PROGRAM P1_04_Alarms
VAR
	iActive				:INT;
	iAck				:INT;
	iRaise				:INT;
	iDisabled			:INT;
	
	bAlarmDisabled		:BOOL;
	
	bAlarmActive		:BOOL;
	bSP_AlarmActive		:BOOL;
	TON_AlarmOK			:TON;
	TON_SP_AlarmOK		:TON;
END_VAR

VAR PERSISTENT
	fbAlarm				:ARRAY [0..69] OF FB_AlarmDiagnostic;
END_VAR

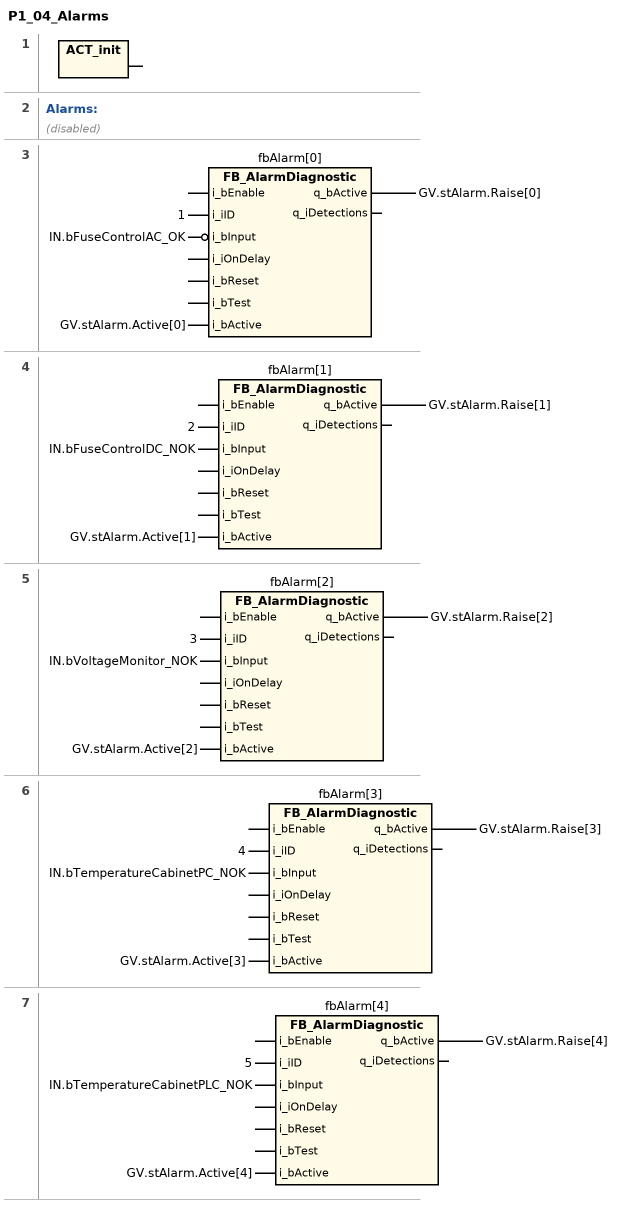
// NETWORK 1
ACT_init();

// NETWORK 2 (disabled)
// label: Alarms

// NETWORK 3
fbAlarm[0](i_iID := 1, i_bInput := NOT IN.bFuseControlAC_OK, i_bActive := GV.stAlarm.Active[0]); // FB_AlarmDiagnostic
GV.stAlarm.Raise[0] := fbAlarm[0].q_bActive;

// NETWORK 4
fbAlarm[1](i_iID := 2, i_bInput := IN.bFuseControlDC_NOK, i_bActive := GV.stAlarm.Active[1]); // FB_AlarmDiagnostic
GV.stAlarm.Raise[1] := fbAlarm[1].q_bActive;

// NETWORK 5
fbAlarm[2](i_iID := 3, i_bInput := IN.bVoltageMonitor_NOK, i_bActive := GV.stAlarm.Active[2]); // FB_AlarmDiagnostic
GV.stAlarm.Raise[2] := fbAlarm[2].q_bActive;

// NETWORK 6
fbAlarm[3](i_iID := 4, i_bInput := IN.bTemperatureCabinetPC_NOK, i_bActive := GV.stAlarm.Active[3]); // FB_AlarmDiagnostic
GV.stAlarm.Raise[3] := fbAlarm[3].q_bActive;

// NETWORK 7
fbAlarm[4](i_iID := 5, i_bInput := IN.bTemperatureCabinetPLC_NOK, i_bActive := GV.stAlarm.Active[4]); // FB_AlarmDiagnostic
GV.stAlarm.Raise[4] := fbAlarm[4].q_bActive;

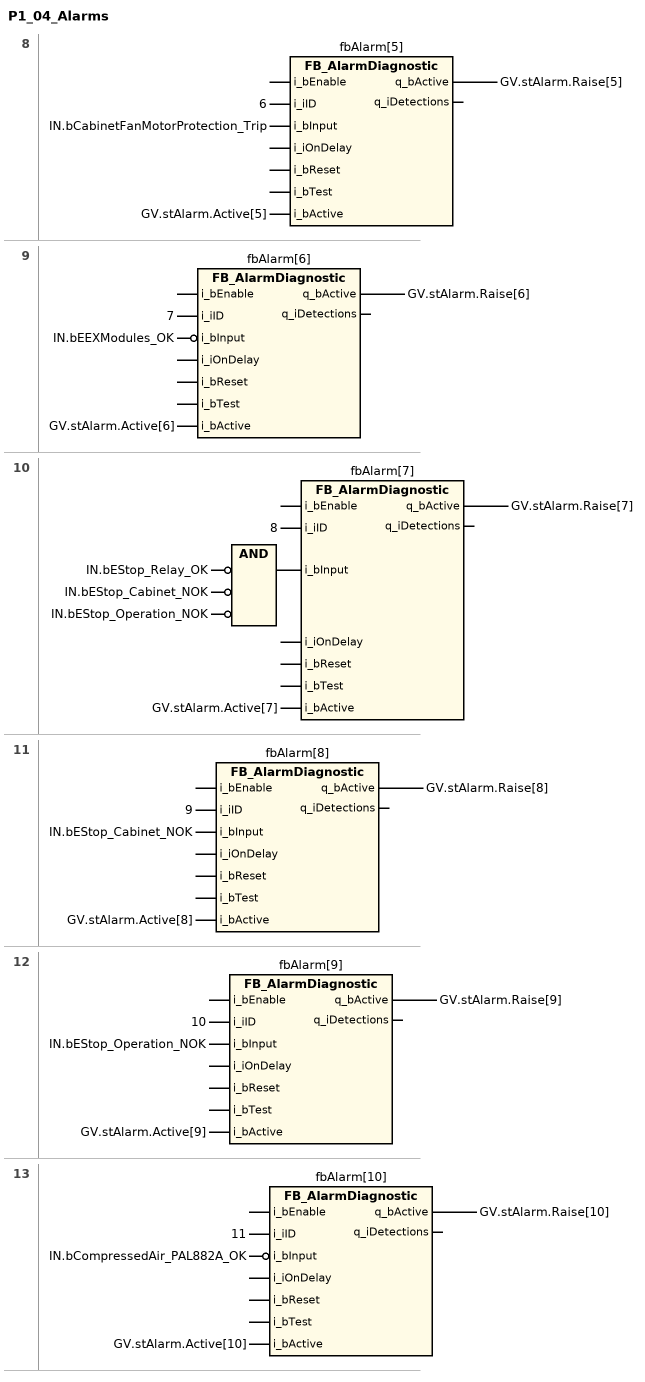
// NETWORK 8
fbAlarm[5](i_iID := 6, i_bInput := IN.bCabinetFanMotorProtection_Trip, i_bActive := GV.stAlarm.Active[5]); // FB_AlarmDiagnostic
GV.stAlarm.Raise[5] := fbAlarm[5].q_bActive;

// NETWORK 9
fbAlarm[6](i_iID := 7, i_bInput := NOT IN.bEEXModules_OK, i_bActive := GV.stAlarm.Active[6]); // FB_AlarmDiagnostic
GV.stAlarm.Raise[6] := fbAlarm[6].q_bActive;

// NETWORK 10
fbAlarm[7](
    i_iID := 8,
    i_bInput := NOT IN.bEStop_Relay_OK AND NOT IN.bEStop_Cabinet_NOK AND NOT IN.bEStop_Operation_NOK,
    i_bActive := GV.stAlarm.Active[7]); // FB_AlarmDiagnostic
GV.stAlarm.Raise[7] := fbAlarm[7].q_bActive;

// NETWORK 11
fbAlarm[8](i_iID := 9, i_bInput := IN.bEStop_Cabinet_NOK, i_bActive := GV.stAlarm.Active[8]); // FB_AlarmDiagnostic
GV.stAlarm.Raise[8] := fbAlarm[8].q_bActive;

// NETWORK 12
fbAlarm[9](i_iID := 10, i_bInput := IN.bEStop_Operation_NOK, i_bActive := GV.stAlarm.Active[9]); // FB_AlarmDiagnostic
GV.stAlarm.Raise[9] := fbAlarm[9].q_bActive;

// NETWORK 13
fbAlarm[10](i_iID := 11, i_bInput := NOT IN.bCompressedAir_PAL882A_OK, i_bActive := GV.stAlarm.Active[10]); // FB_AlarmDiagnostic
GV.stAlarm.Raise[10] := fbAlarm[10].q_bActive;

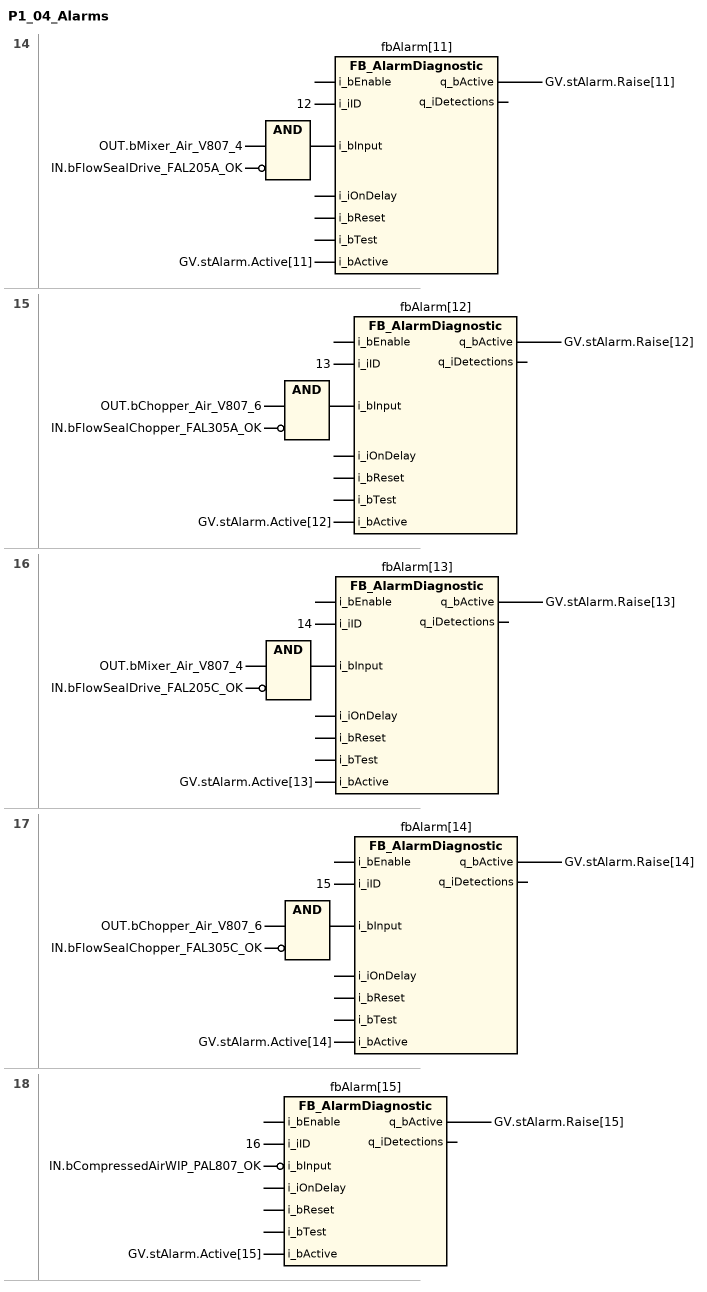
// NETWORK 14
fbAlarm[11](
    i_iID := 12,
    i_bInput := OUT.bMixer_Air_V807_4 AND NOT IN.bFlowSealDrive_FAL205A_OK,
    i_bActive := GV.stAlarm.Active[11]); // FB_AlarmDiagnostic
GV.stAlarm.Raise[11] := fbAlarm[11].q_bActive;

// NETWORK 15
fbAlarm[12](
    i_iID := 13,
    i_bInput := OUT.bChopper_Air_V807_6 AND NOT IN.bFlowSealChopper_FAL305A_OK,
    i_bActive := GV.stAlarm.Active[12]); // FB_AlarmDiagnostic
GV.stAlarm.Raise[12] := fbAlarm[12].q_bActive;

// NETWORK 16
fbAlarm[13](
    i_iID := 14,
    i_bInput := OUT.bMixer_Air_V807_4 AND NOT IN.bFlowSealDrive_FAL205C_OK,
    i_bActive := GV.stAlarm.Active[13]); // FB_AlarmDiagnostic
GV.stAlarm.Raise[13] := fbAlarm[13].q_bActive;

// NETWORK 17
fbAlarm[14](
    i_iID := 15,
    i_bInput := OUT.bChopper_Air_V807_6 AND NOT IN.bFlowSealChopper_FAL305C_OK,
    i_bActive := GV.stAlarm.Active[14]); // FB_AlarmDiagnostic
GV.stAlarm.Raise[14] := fbAlarm[14].q_bActive;

// NETWORK 18
fbAlarm[15](i_iID := 16, i_bInput := NOT IN.bCompressedAirWIP_PAL807_OK, i_bActive := GV.stAlarm.Active[15]); // FB_AlarmDiagnostic
GV.stAlarm.Raise[15] := fbAlarm[15].q_bActive;

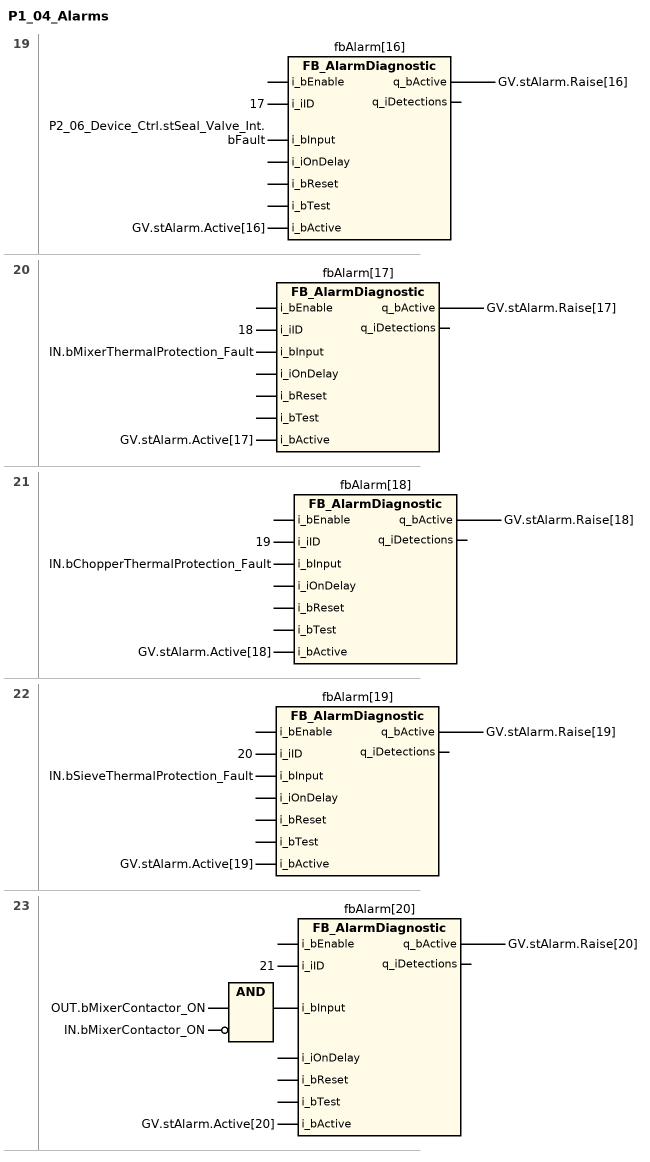
// NETWORK 19
fbAlarm[16](
    i_iID := 17,
    i_bInput := P2_06_Device_Ctrl.stSeal_Valve_Int.bFault,
    i_bActive := GV.stAlarm.Active[16]); // FB_AlarmDiagnostic
GV.stAlarm.Raise[16] := fbAlarm[16].q_bActive;

// NETWORK 20
fbAlarm[17](i_iID := 18, i_bInput := IN.bMixerThermalProtection_Fault, i_bActive := GV.stAlarm.Active[17]); // FB_AlarmDiagnostic
GV.stAlarm.Raise[17] := fbAlarm[17].q_bActive;

// NETWORK 21
fbAlarm[18](i_iID := 19, i_bInput := IN.bChopperThermalProtection_Fault, i_bActive := GV.stAlarm.Active[18]); // FB_AlarmDiagnostic
GV.stAlarm.Raise[18] := fbAlarm[18].q_bActive;

// NETWORK 22
fbAlarm[19](i_iID := 20, i_bInput := IN.bSieveThermalProtection_Fault, i_bActive := GV.stAlarm.Active[19]); // FB_AlarmDiagnostic
GV.stAlarm.Raise[19] := fbAlarm[19].q_bActive;

// NETWORK 23
fbAlarm[20](
    i_iID := 21,
    i_bInput := OUT.bMixerContactor_ON AND NOT IN.bMixerContactor_ON,
    i_bActive := GV.stAlarm.Active[20]); // FB_AlarmDiagnostic
GV.stAlarm.Raise[20] := fbAlarm[20].q_bActive;

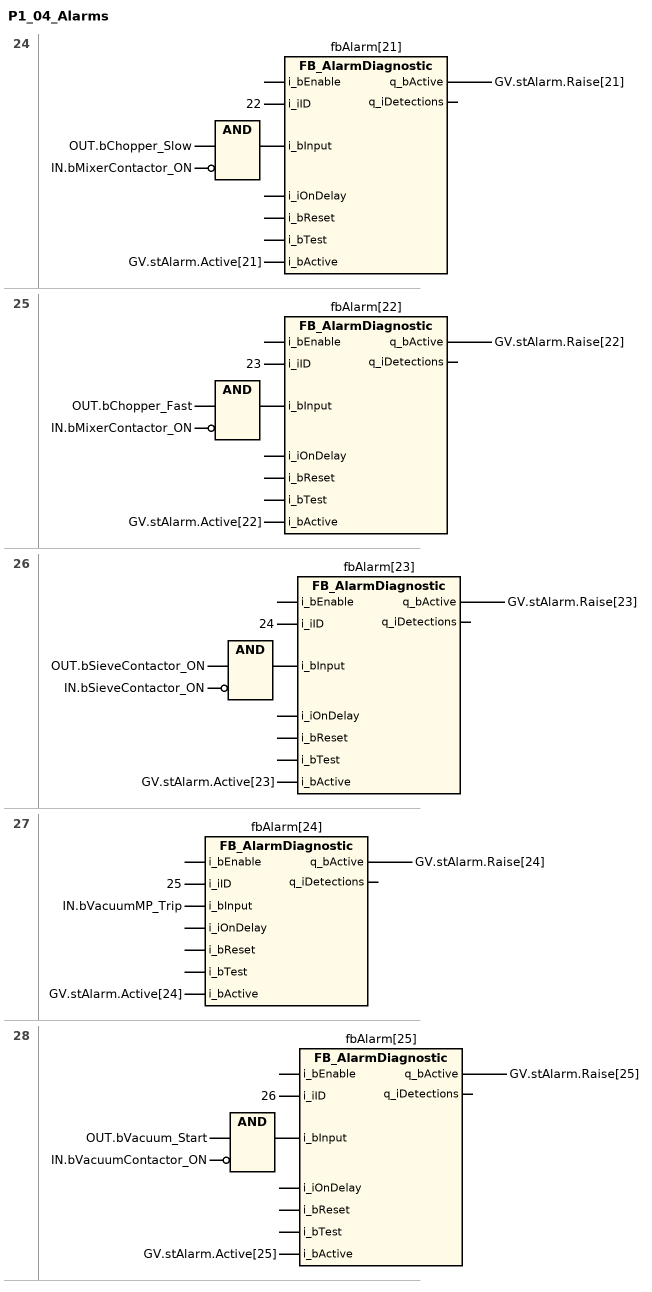
// NETWORK 24
fbAlarm[21](
    i_iID := 22,
    i_bInput := OUT.bChopper_Slow AND NOT IN.bMixerContactor_ON,
    i_bActive := GV.stAlarm.Active[21]); // FB_AlarmDiagnostic
GV.stAlarm.Raise[21] := fbAlarm[21].q_bActive;

// NETWORK 25
fbAlarm[22](
    i_iID := 23,
    i_bInput := OUT.bChopper_Fast AND NOT IN.bMixerContactor_ON,
    i_bActive := GV.stAlarm.Active[22]); // FB_AlarmDiagnostic
GV.stAlarm.Raise[22] := fbAlarm[22].q_bActive;

// NETWORK 26
fbAlarm[23](
    i_iID := 24,
    i_bInput := OUT.bSieveContactor_ON AND NOT IN.bSieveContactor_ON,
    i_bActive := GV.stAlarm.Active[23]); // FB_AlarmDiagnostic
GV.stAlarm.Raise[23] := fbAlarm[23].q_bActive;

// NETWORK 27
fbAlarm[24](i_iID := 25, i_bInput := IN.bVacuumMP_Trip, i_bActive := GV.stAlarm.Active[24]); // FB_AlarmDiagnostic
GV.stAlarm.Raise[24] := fbAlarm[24].q_bActive;

// NETWORK 28
fbAlarm[25](
    i_iID := 26,
    i_bInput := OUT.bVacuum_Start AND NOT IN.bVacuumContactor_ON,
    i_bActive := GV.stAlarm.Active[25]); // FB_AlarmDiagnostic
GV.stAlarm.Raise[25] := fbAlarm[25].q_bActive;

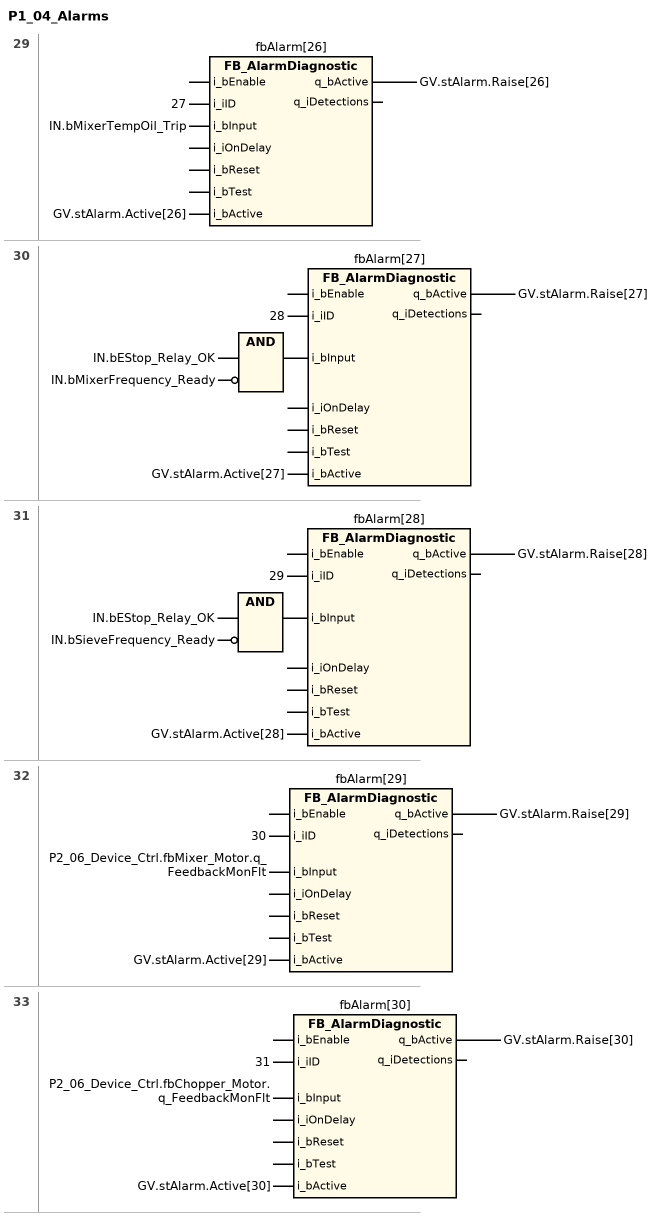
// NETWORK 29
fbAlarm[26](i_iID := 27, i_bInput := IN.bMixerTempOil_Trip, i_bActive := GV.stAlarm.Active[26]); // FB_AlarmDiagnostic
GV.stAlarm.Raise[26] := fbAlarm[26].q_bActive;

// NETWORK 30
fbAlarm[27](
    i_iID := 28,
    i_bInput := IN.bEStop_Relay_OK AND NOT IN.bMixerFrequency_Ready,
    i_bActive := GV.stAlarm.Active[27]); // FB_AlarmDiagnostic
GV.stAlarm.Raise[27] := fbAlarm[27].q_bActive;

// NETWORK 31
fbAlarm[28](
    i_iID := 29,
    i_bInput := IN.bEStop_Relay_OK AND NOT IN.bSieveFrequency_Ready,
    i_bActive := GV.stAlarm.Active[28]); // FB_AlarmDiagnostic
GV.stAlarm.Raise[28] := fbAlarm[28].q_bActive;

// NETWORK 32
fbAlarm[29](
    i_iID := 30,
    i_bInput := P2_06_Device_Ctrl.fbMixer_Motor.q_FeedbackMonFlt,
    i_bActive := GV.stAlarm.Active[29]); // FB_AlarmDiagnostic
GV.stAlarm.Raise[29] := fbAlarm[29].q_bActive;

// NETWORK 33
fbAlarm[30](
    i_iID := 31,
    i_bInput := P2_06_Device_Ctrl.fbChopper_Motor.q_FeedbackMonFlt,
    i_bActive := GV.stAlarm.Active[30]); // FB_AlarmDiagnostic
GV.stAlarm.Raise[30] := fbAlarm[30].q_bActive;

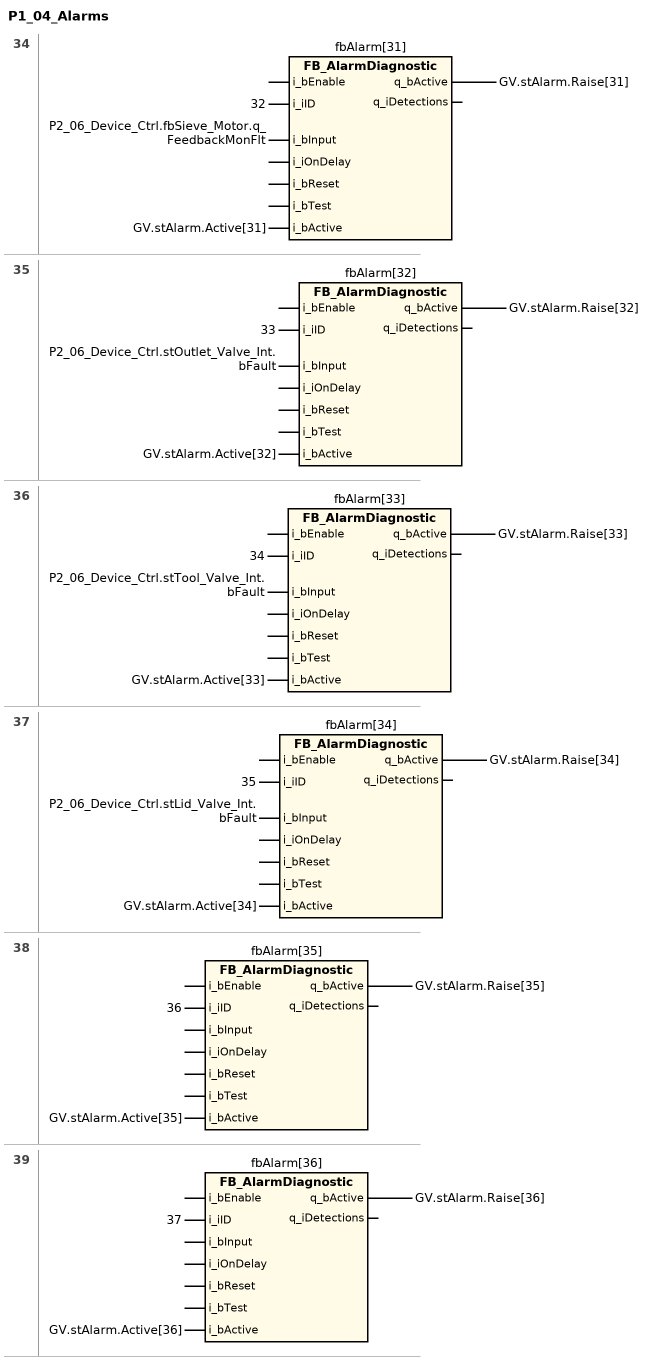
// NETWORK 34
fbAlarm[31](
    i_iID := 32,
    i_bInput := P2_06_Device_Ctrl.fbSieve_Motor.q_FeedbackMonFlt,
    i_bActive := GV.stAlarm.Active[31]); // FB_AlarmDiagnostic
GV.stAlarm.Raise[31] := fbAlarm[31].q_bActive;

// NETWORK 35
fbAlarm[32](
    i_iID := 33,
    i_bInput := P2_06_Device_Ctrl.stOutlet_Valve_Int.bFault,
    i_bActive := GV.stAlarm.Active[32]); // FB_AlarmDiagnostic
GV.stAlarm.Raise[32] := fbAlarm[32].q_bActive;

// NETWORK 36
fbAlarm[33](
    i_iID := 34,
    i_bInput := P2_06_Device_Ctrl.stTool_Valve_Int.bFault,
    i_bActive := GV.stAlarm.Active[33]); // FB_AlarmDiagnostic
GV.stAlarm.Raise[33] := fbAlarm[33].q_bActive;

// NETWORK 37
fbAlarm[34](
    i_iID := 35,
    i_bInput := P2_06_Device_Ctrl.stLid_Valve_Int.bFault,
    i_bActive := GV.stAlarm.Active[34]); // FB_AlarmDiagnostic
GV.stAlarm.Raise[34] := fbAlarm[34].q_bActive;

// NETWORK 38
fbAlarm[35](i_iID := 36, i_bActive := GV.stAlarm.Active[35]); // FB_AlarmDiagnostic
GV.stAlarm.Raise[35] := fbAlarm[35].q_bActive;

// NETWORK 39
fbAlarm[36](i_iID := 37, i_bActive := GV.stAlarm.Active[36]); // FB_AlarmDiagnostic
GV.stAlarm.Raise[36] := fbAlarm[36].q_bActive;

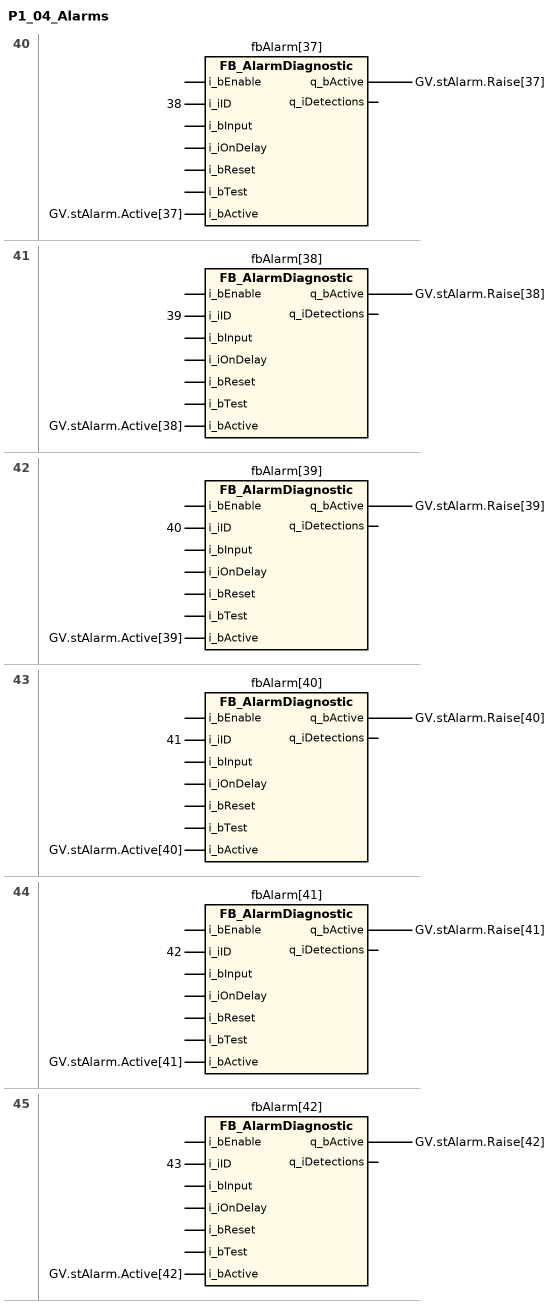
// NETWORK 40
fbAlarm[37](i_iID := 38, i_bActive := GV.stAlarm.Active[37]); // FB_AlarmDiagnostic
GV.stAlarm.Raise[37] := fbAlarm[37].q_bActive;

// NETWORK 41
fbAlarm[38](i_iID := 39, i_bActive := GV.stAlarm.Active[38]); // FB_AlarmDiagnostic
GV.stAlarm.Raise[38] := fbAlarm[38].q_bActive;

// NETWORK 42
fbAlarm[39](i_iID := 40, i_bActive := GV.stAlarm.Active[39]); // FB_AlarmDiagnostic
GV.stAlarm.Raise[39] := fbAlarm[39].q_bActive;

// NETWORK 43
fbAlarm[40](i_iID := 41, i_bActive := GV.stAlarm.Active[40]); // FB_AlarmDiagnostic
GV.stAlarm.Raise[40] := fbAlarm[40].q_bActive;

// NETWORK 44
fbAlarm[41](i_iID := 42, i_bActive := GV.stAlarm.Active[41]); // FB_AlarmDiagnostic
GV.stAlarm.Raise[41] := fbAlarm[41].q_bActive;

// NETWORK 45
fbAlarm[42](i_iID := 43, i_bActive := GV.stAlarm.Active[42]); // FB_AlarmDiagnostic
GV.stAlarm.Raise[42] := fbAlarm[42].q_bActive;

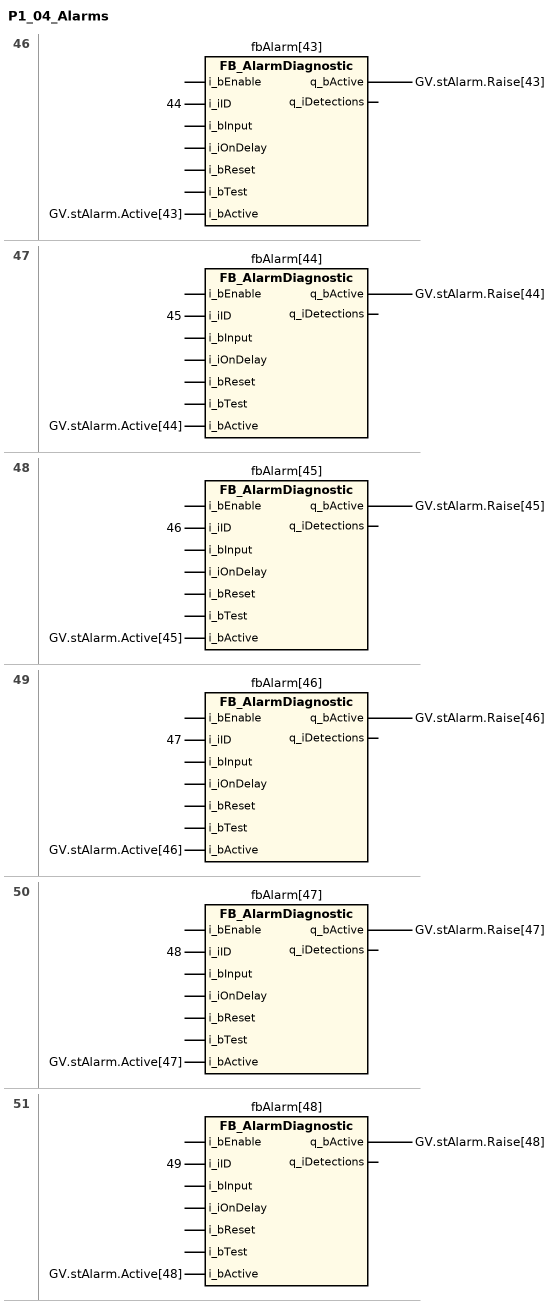
// NETWORK 46
fbAlarm[43](i_iID := 44, i_bActive := GV.stAlarm.Active[43]); // FB_AlarmDiagnostic
GV.stAlarm.Raise[43] := fbAlarm[43].q_bActive;

// NETWORK 47
fbAlarm[44](i_iID := 45, i_bActive := GV.stAlarm.Active[44]); // FB_AlarmDiagnostic
GV.stAlarm.Raise[44] := fbAlarm[44].q_bActive;

// NETWORK 48
fbAlarm[45](i_iID := 46, i_bActive := GV.stAlarm.Active[45]); // FB_AlarmDiagnostic
GV.stAlarm.Raise[45] := fbAlarm[45].q_bActive;

// NETWORK 49
fbAlarm[46](i_iID := 47, i_bActive := GV.stAlarm.Active[46]); // FB_AlarmDiagnostic
GV.stAlarm.Raise[46] := fbAlarm[46].q_bActive;

// NETWORK 50
fbAlarm[47](i_iID := 48, i_bActive := GV.stAlarm.Active[47]); // FB_AlarmDiagnostic
GV.stAlarm.Raise[47] := fbAlarm[47].q_bActive;

// NETWORK 51
fbAlarm[48](i_iID := 49, i_bActive := GV.stAlarm.Active[48]); // FB_AlarmDiagnostic
GV.stAlarm.Raise[48] := fbAlarm[48].q_bActive;

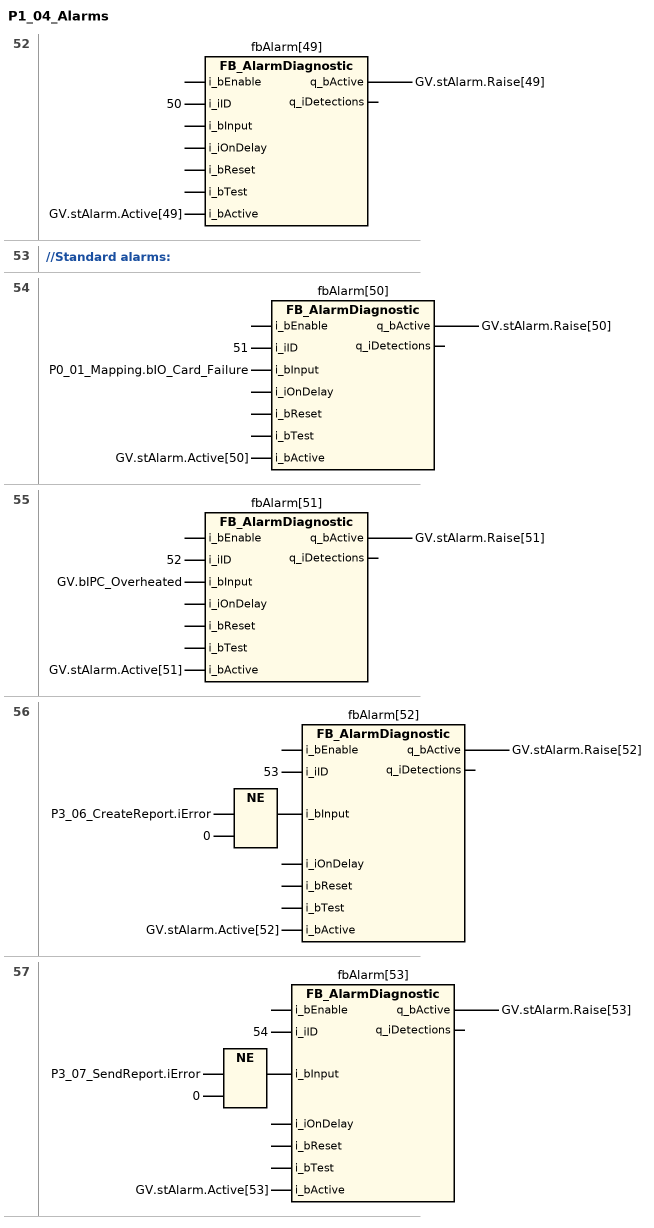
// NETWORK 52
fbAlarm[49](i_iID := 50, i_bActive := GV.stAlarm.Active[49]); // FB_AlarmDiagnostic
GV.stAlarm.Raise[49] := fbAlarm[49].q_bActive;

// NETWORK 53
// label: //Standard alarms

// NETWORK 54
fbAlarm[50](i_iID := 51, i_bInput := P0_01_Mapping.bIO_Card_Failure, i_bActive := GV.stAlarm.Active[50]); // FB_AlarmDiagnostic
GV.stAlarm.Raise[50] := fbAlarm[50].q_bActive;

// NETWORK 55
fbAlarm[51](i_iID := 52, i_bInput := GV.bIPC_Overheated, i_bActive := GV.stAlarm.Active[51]); // FB_AlarmDiagnostic
GV.stAlarm.Raise[51] := fbAlarm[51].q_bActive;

// NETWORK 56
fbAlarm[52](i_iID := 53, i_bInput := P3_06_CreateReport.iError <> 0, i_bActive := GV.stAlarm.Active[52]); // FB_AlarmDiagnostic
GV.stAlarm.Raise[52] := fbAlarm[52].q_bActive;

// NETWORK 57
fbAlarm[53](i_iID := 54, i_bInput := P3_07_SendReport.iError <> 0, i_bActive := GV.stAlarm.Active[53]); // FB_AlarmDiagnostic
GV.stAlarm.Raise[53] := fbAlarm[53].q_bActive;

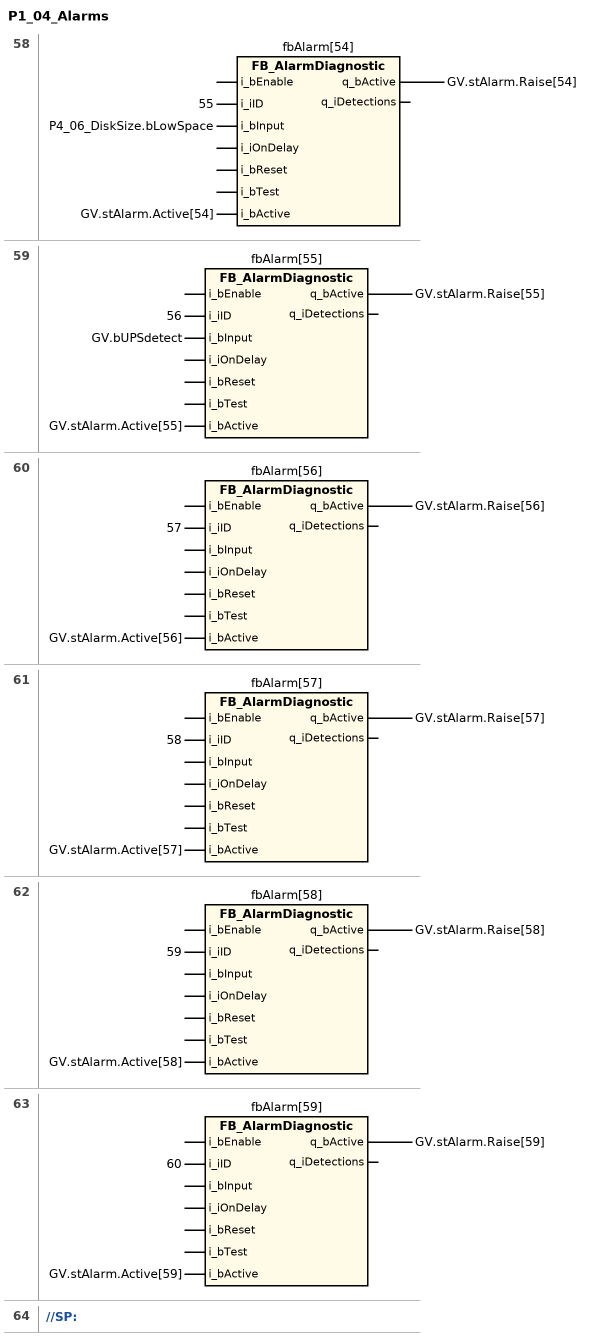
// NETWORK 58
fbAlarm[54](i_iID := 55, i_bInput := P4_06_DiskSize.bLowSpace, i_bActive := GV.stAlarm.Active[54]); // FB_AlarmDiagnostic
GV.stAlarm.Raise[54] := fbAlarm[54].q_bActive;

// NETWORK 59
fbAlarm[55](i_iID := 56, i_bInput := GV.bUPSdetect, i_bActive := GV.stAlarm.Active[55]); // FB_AlarmDiagnostic
GV.stAlarm.Raise[55] := fbAlarm[55].q_bActive;

// NETWORK 60
fbAlarm[56](i_iID := 57, i_bActive := GV.stAlarm.Active[56]); // FB_AlarmDiagnostic
GV.stAlarm.Raise[56] := fbAlarm[56].q_bActive;

// NETWORK 61
fbAlarm[57](i_iID := 58, i_bActive := GV.stAlarm.Active[57]); // FB_AlarmDiagnostic
GV.stAlarm.Raise[57] := fbAlarm[57].q_bActive;

// NETWORK 62
fbAlarm[58](i_iID := 59, i_bActive := GV.stAlarm.Active[58]); // FB_AlarmDiagnostic
GV.stAlarm.Raise[58] := fbAlarm[58].q_bActive;

// NETWORK 63
fbAlarm[59](i_iID := 60, i_bActive := GV.stAlarm.Active[59]); // FB_AlarmDiagnostic
GV.stAlarm.Raise[59] := fbAlarm[59].q_bActive;

// NETWORK 64
// label: //SP

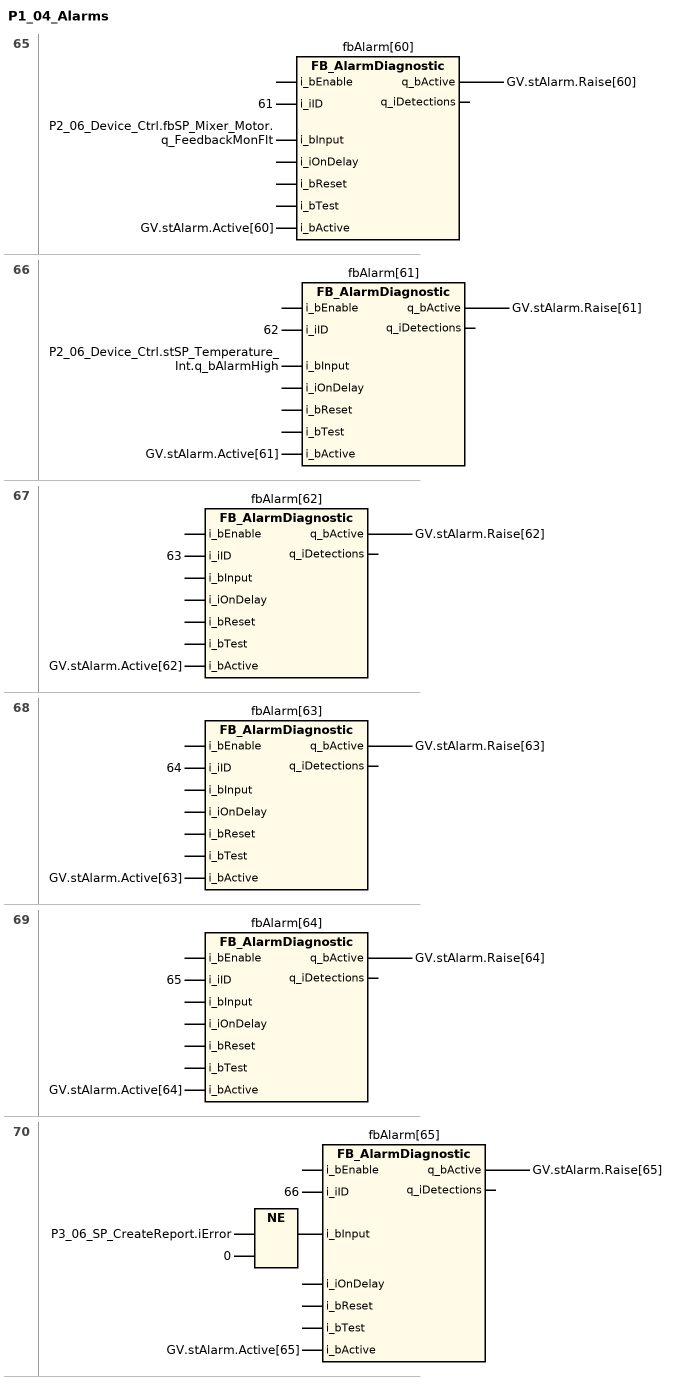
// NETWORK 65
fbAlarm[60](
    i_iID := 61,
    i_bInput := P2_06_Device_Ctrl.fbSP_Mixer_Motor.q_FeedbackMonFlt,
    i_bActive := GV.stAlarm.Active[60]); // FB_AlarmDiagnostic
GV.stAlarm.Raise[60] := fbAlarm[60].q_bActive;

// NETWORK 66
fbAlarm[61](
    i_iID := 62,
    i_bInput := P2_06_Device_Ctrl.stSP_Temperature_Int.q_bAlarmHigh,
    i_bActive := GV.stAlarm.Active[61]); // FB_AlarmDiagnostic
GV.stAlarm.Raise[61] := fbAlarm[61].q_bActive;

// NETWORK 67
fbAlarm[62](i_iID := 63, i_bActive := GV.stAlarm.Active[62]); // FB_AlarmDiagnostic
GV.stAlarm.Raise[62] := fbAlarm[62].q_bActive;

// NETWORK 68
fbAlarm[63](i_iID := 64, i_bActive := GV.stAlarm.Active[63]); // FB_AlarmDiagnostic
GV.stAlarm.Raise[63] := fbAlarm[63].q_bActive;

// NETWORK 69
fbAlarm[64](i_iID := 65, i_bActive := GV.stAlarm.Active[64]); // FB_AlarmDiagnostic
GV.stAlarm.Raise[64] := fbAlarm[64].q_bActive;

// NETWORK 70
fbAlarm[65](i_iID := 66, i_bInput := P3_06_SP_CreateReport.iError <> 0, i_bActive := GV.stAlarm.Active[65]); // FB_AlarmDiagnostic
GV.stAlarm.Raise[65] := fbAlarm[65].q_bActive;

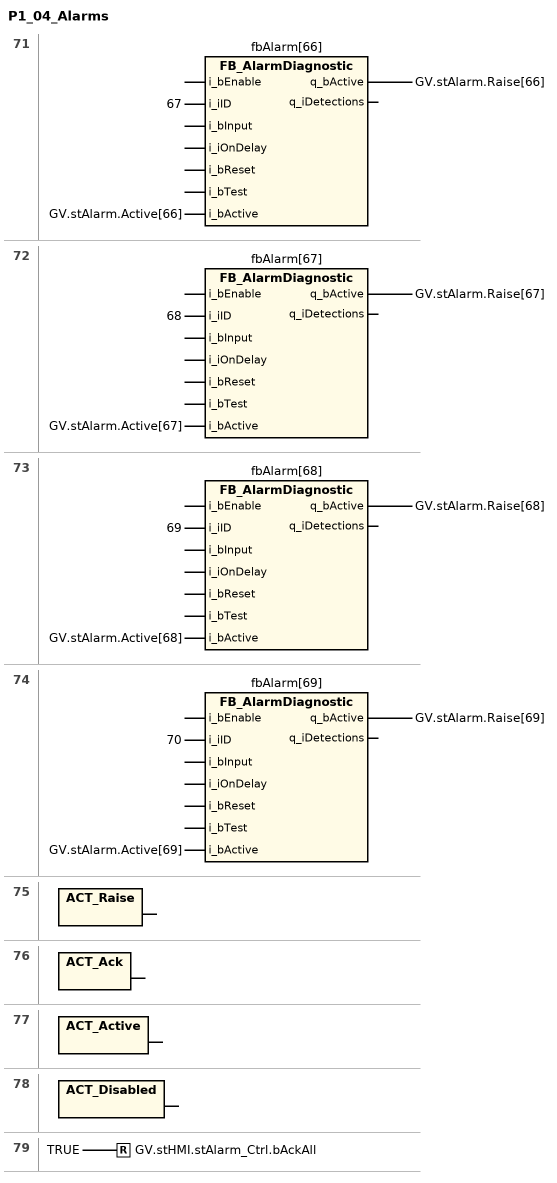
// NETWORK 71
fbAlarm[66](i_iID := 67, i_bActive := GV.stAlarm.Active[66]); // FB_AlarmDiagnostic
GV.stAlarm.Raise[66] := fbAlarm[66].q_bActive;

// NETWORK 72
fbAlarm[67](i_iID := 68, i_bActive := GV.stAlarm.Active[67]); // FB_AlarmDiagnostic
GV.stAlarm.Raise[67] := fbAlarm[67].q_bActive;

// NETWORK 73
fbAlarm[68](i_iID := 69, i_bActive := GV.stAlarm.Active[68]); // FB_AlarmDiagnostic
GV.stAlarm.Raise[68] := fbAlarm[68].q_bActive;

// NETWORK 74
fbAlarm[69](i_iID := 70, i_bActive := GV.stAlarm.Active[69]); // FB_AlarmDiagnostic
GV.stAlarm.Raise[69] := fbAlarm[69].q_bActive;

// NETWORK 75
ACT_Raise();

// NETWORK 76
ACT_Ack();

// NETWORK 77
ACT_Active();

// NETWORK 78
ACT_Disabled();

// NETWORK 79
GV.stHMI.stAlarm_Ctrl.bAckAll R= TRUE;

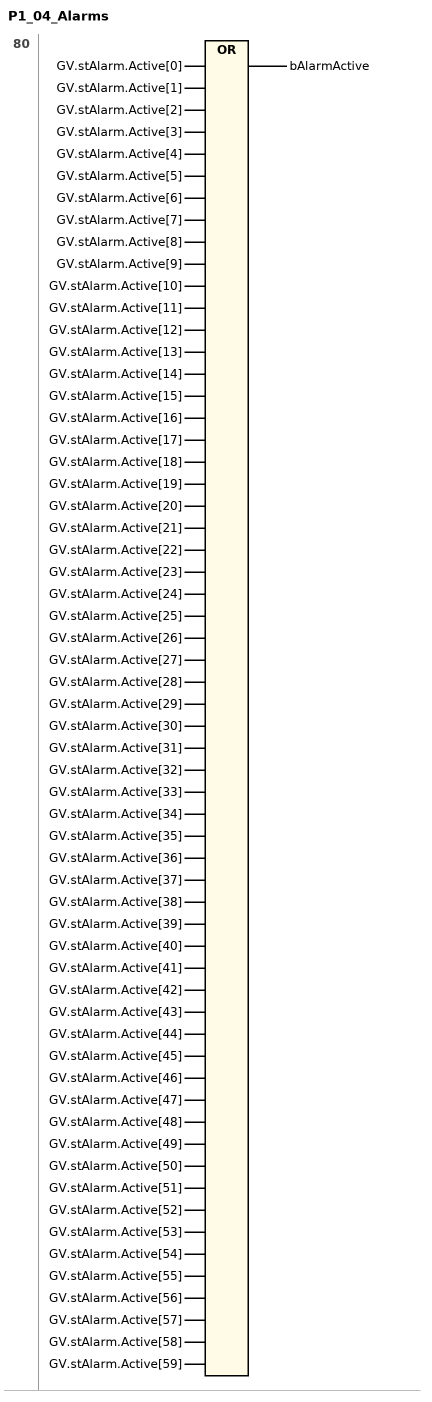
// NETWORK 80
bAlarmActive := GV.stAlarm.Active[0] OR GV.stAlarm.Active[1] OR GV.stAlarm.Active[2] OR GV.stAlarm.Active[3] OR GV.stAlarm.Active[4] OR GV.stAlarm.Active[5] OR GV.stAlarm.Active[6] OR GV.stAlarm.Active[7] OR GV.stAlarm.Active[8] OR GV.stAlarm.Active[9] OR GV.stAlarm.Active[10] OR GV.stAlarm.Active[11] OR GV.stAlarm.Active[12] OR GV.stAlarm.Active[13] OR GV.stAlarm.Active[14] OR GV.stAlarm.Active[15] OR GV.stAlarm.Active[16] OR GV.stAlarm.Active[17] OR GV.stAlarm.Active[18] OR GV.stAlarm.Active[19] OR GV.stAlarm.Active[20] OR GV.stAlarm.Active[21] OR GV.stAlarm.Active[22] OR GV.stAlarm.Active[23] OR GV.stAlarm.Active[24] OR GV.stAlarm.Active[25] OR GV.stAlarm.Active[26] OR GV.stAlarm.Active[27] OR GV.stAlarm.Active[28] OR GV.stAlarm.Active[29] OR GV.stAlarm.Active[30] OR GV.stAlarm.Active[31] OR GV.stAlarm.Active[32] OR GV.stAlarm.Active[33] OR GV.stAlarm.Active[34] OR GV.stAlarm.Active[35] OR GV.stAlarm.Active[36] OR GV.stAlarm.Active[37] OR GV.stAlarm.Active[38] OR GV.stAlarm.Active[39] OR GV.stAlarm.Active[40] OR GV.stAlarm.Active[41] OR GV.stAlarm.Active[42] OR GV.stAlarm.Active[43] OR GV.stAlarm.Active[44] OR GV.stAlarm.Active[45] OR GV.stAlarm.Active[46] OR GV.stAlarm.Active[47] OR GV.stAlarm.Active[48] OR GV.stAlarm.Active[49] OR GV.stAlarm.Active[50] OR GV.stAlarm.Active[51] OR GV.stAlarm.Active[52] OR GV.stAlarm.Active[53] OR GV.stAlarm.Active[54] OR GV.stAlarm.Active[55] OR GV.stAlarm.Active[56] OR GV.stAlarm.Active[57] OR GV.stAlarm.Active[58] OR GV.stAlarm.Active[59];

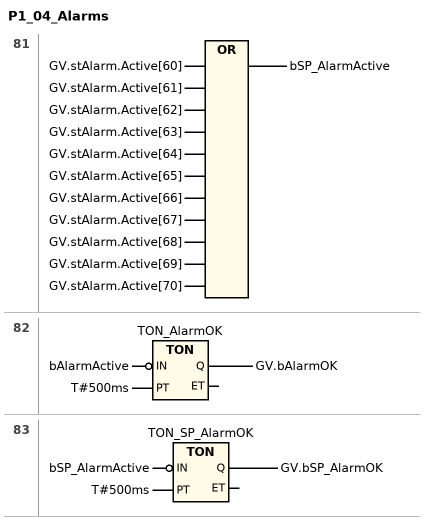
// NETWORK 81
bSP_AlarmActive := GV.stAlarm.Active[60] OR GV.stAlarm.Active[61] OR GV.stAlarm.Active[62] OR GV.stAlarm.Active[63] OR GV.stAlarm.Active[64] OR GV.stAlarm.Active[65] OR GV.stAlarm.Active[66] OR GV.stAlarm.Active[67] OR GV.stAlarm.Active[68] OR GV.stAlarm.Active[69] OR GV.stAlarm.Active[70];

// NETWORK 82
TON_AlarmOK(IN := NOT bAlarmActive, PT := T#500ms); // TON
GV.bAlarmOK := TON_AlarmOK.Q;

// NETWORK 83
TON_SP_AlarmOK(IN := NOT bSP_AlarmActive, PT := T#500ms); // TON
GV.bSP_AlarmOK := TON_SP_AlarmOK.Q;

ACTION ACT_Ack:
FOR iAck:=0 TO 69 DO
	IF GV.stAlarm.Alarm[iAck].eConfirmationState = 3 OR GV.stHMI.stAlarm_Ctrl.bAckAll THEN
		GV.stAlarm.Alarm[iAck].Clear(0,1);
	END_IF
	
END_FOR
END_ACTION

ACTION ACT_Active:
FOR iActive:=0 TO 69 DO
	GV.stAlarm.Active[iActive]:=GV.stAlarm.Alarm[iActive].bActive;
END_FOR
END_ACTION

ACTION ACT_Disabled:
bAlarmDisabled:=FALSE;
FOR iDisabled:=0 TO 69 DO
	IF NOT fbAlarm[iDisabled].i_bEnable THEN
		bAlarmDisabled:=TRUE;
	END_IF
END_FOR
END_ACTION

ACTION ACT_Init:
IF MAIN.bFirstCycle THEN
	//Critical
	GV.stAlarm.Alarm[0].CreateEx(TC_EVENTS.Alarms.AlarmsEvent1,1,0);
	GV.stAlarm.Alarm[1].CreateEx(TC_EVENTS.Alarms.AlarmsEvent2,1,0);
	GV.stAlarm.Alarm[2].CreateEx(TC_EVENTS.Alarms.AlarmsEvent3,1,0);
	GV.stAlarm.Alarm[3].CreateEx(TC_EVENTS.Alarms.AlarmsEvent4,1,0);
	GV.stAlarm.Alarm[4].CreateEx(TC_EVENTS.Alarms.AlarmsEvent5,1,0);
	GV.stAlarm.Alarm[5].CreateEx(TC_EVENTS.Alarms.AlarmsEvent6,1,0);
	GV.stAlarm.Alarm[6].CreateEx(TC_EVENTS.Alarms.AlarmsEvent7,1,0);
	GV.stAlarm.Alarm[7].CreateEx(TC_EVENTS.Alarms.AlarmsEvent8,1,0);
	GV.stAlarm.Alarm[8].CreateEx(TC_EVENTS.Alarms.AlarmsEvent9,1,0);
	GV.stAlarm.Alarm[9].CreateEx(TC_EVENTS.Alarms.AlarmsEvent10,1,0);
	GV.stAlarm.Alarm[10].CreateEx(TC_EVENTS.Alarms.AlarmsEvent11,1,0);
	GV.stAlarm.Alarm[11].CreateEx(TC_EVENTS.Alarms.AlarmsEvent12,1,0);
	GV.stAlarm.Alarm[12].CreateEx(TC_EVENTS.Alarms.AlarmsEvent13,1,0);
	GV.stAlarm.Alarm[13].CreateEx(TC_EVENTS.Alarms.AlarmsEvent14,1,0);
	GV.stAlarm.Alarm[14].CreateEx(TC_EVENTS.Alarms.AlarmsEvent15,1,0);
	GV.stAlarm.Alarm[15].CreateEx(TC_EVENTS.Alarms.AlarmsEvent16,1,0);
	GV.stAlarm.Alarm[16].CreateEx(TC_EVENTS.Alarms.AlarmsEvent17,1,0);
	GV.stAlarm.Alarm[17].CreateEx(TC_EVENTS.Alarms.AlarmsEvent18,1,0);
	GV.stAlarm.Alarm[18].CreateEx(TC_EVENTS.Alarms.AlarmsEvent19,1,0);
	GV.stAlarm.Alarm[19].CreateEx(TC_EVENTS.Alarms.AlarmsEvent20,1,0);
	GV.stAlarm.Alarm[20].CreateEx(TC_EVENTS.Alarms.AlarmsEvent21,1,0);
	GV.stAlarm.Alarm[21].CreateEx(TC_EVENTS.Alarms.AlarmsEvent22,1,0);
	GV.stAlarm.Alarm[22].CreateEx(TC_EVENTS.Alarms.AlarmsEvent23,1,0);
	GV.stAlarm.Alarm[23].CreateEx(TC_EVENTS.Alarms.AlarmsEvent24,1,0);
	GV.stAlarm.Alarm[24].CreateEx(TC_EVENTS.Alarms.AlarmsEvent25,1,0);
	GV.stAlarm.Alarm[25].CreateEx(TC_EVENTS.Alarms.AlarmsEvent26,1,0);
	GV.stAlarm.Alarm[26].CreateEx(TC_EVENTS.Alarms.AlarmsEvent27,1,0);
	GV.stAlarm.Alarm[27].CreateEx(TC_EVENTS.Alarms.AlarmsEvent28,1,0);
	GV.stAlarm.Alarm[28].CreateEx(TC_EVENTS.Alarms.AlarmsEvent29,1,0);
	GV.stAlarm.Alarm[29].CreateEx(TC_EVENTS.Alarms.AlarmsEvent30,1,0);
	GV.stAlarm.Alarm[30].CreateEx(TC_EVENTS.Alarms.AlarmsEvent31,1,0);
	GV.stAlarm.Alarm[31].CreateEx(TC_EVENTS.Alarms.AlarmsEvent32,1,0);
	GV.stAlarm.Alarm[32].CreateEx(TC_EVENTS.Alarms.AlarmsEvent33,1,0);
	GV.stAlarm.Alarm[33].CreateEx(TC_EVENTS.Alarms.AlarmsEvent34,1,0);
	GV.stAlarm.Alarm[34].CreateEx(TC_EVENTS.Alarms.AlarmsEvent35,1,0);
	GV.stAlarm.Alarm[35].CreateEx(TC_EVENTS.Alarms.AlarmsEvent36,1,0);
	GV.stAlarm.Alarm[36].CreateEx(TC_EVENTS.Alarms.AlarmsEvent37,1,0);
	GV.stAlarm.Alarm[37].CreateEx(TC_EVENTS.Alarms.AlarmsEvent38,1,0);
	GV.stAlarm.Alarm[38].CreateEx(TC_EVENTS.Alarms.AlarmsEvent39,1,0);
	GV.stAlarm.Alarm[39].CreateEx(TC_EVENTS.Alarms.AlarmsEvent40,1,0);	
	GV.stAlarm.Alarm[40].CreateEx(TC_EVENTS.Alarms.AlarmsEvent41,1,0);
	GV.stAlarm.Alarm[41].CreateEx(TC_EVENTS.Alarms.AlarmsEvent42,1,0);
	GV.stAlarm.Alarm[42].CreateEx(TC_EVENTS.Alarms.AlarmsEvent43,1,0);
	GV.stAlarm.Alarm[43].CreateEx(TC_EVENTS.Alarms.AlarmsEvent44,1,0);
	GV.stAlarm.Alarm[44].CreateEx(TC_EVENTS.Alarms.AlarmsEvent45,1,0);
	GV.stAlarm.Alarm[45].CreateEx(TC_EVENTS.Alarms.AlarmsEvent46,1,0);
	GV.stAlarm.Alarm[46].CreateEx(TC_EVENTS.Alarms.AlarmsEvent47,1,0);
	GV.stAlarm.Alarm[47].CreateEx(TC_EVENTS.Alarms.AlarmsEvent48,1,0);
	GV.stAlarm.Alarm[48].CreateEx(TC_EVENTS.Alarms.AlarmsEvent49,1,0);
	GV.stAlarm.Alarm[49].CreateEx(TC_EVENTS.Alarms.AlarmsEvent50,1,0);
	GV.stAlarm.Alarm[50].CreateEx(TC_EVENTS.Alarms.AlarmsEvent51,1,0);
	GV.stAlarm.Alarm[51].CreateEx(TC_EVENTS.Alarms.AlarmsEvent52,1,0);
	GV.stAlarm.Alarm[52].CreateEx(TC_EVENTS.Alarms.AlarmsEvent53,1,0);
	GV.stAlarm.Alarm[53].CreateEx(TC_EVENTS.Alarms.AlarmsEvent54,1,0);
	GV.stAlarm.Alarm[54].CreateEx(TC_EVENTS.Alarms.AlarmsEvent55,1,0);
	GV.stAlarm.Alarm[55].CreateEx(TC_EVENTS.Alarms.AlarmsEvent56,1,0);
	GV.stAlarm.Alarm[56].CreateEx(TC_EVENTS.Alarms.AlarmsEvent57,1,0);
	GV.stAlarm.Alarm[57].CreateEx(TC_EVENTS.Alarms.AlarmsEvent58,1,0);
	GV.stAlarm.Alarm[58].CreateEx(TC_EVENTS.Alarms.AlarmsEvent59,1,0);
	GV.stAlarm.Alarm[59].CreateEx(TC_EVENTS.Alarms.AlarmsEvent60,1,0);
	//SP
	GV.stAlarm.Alarm[60].CreateEx(TC_EVENTS.Alarms.AlarmsEvent61,1,0);
	GV.stAlarm.Alarm[61].CreateEx(TC_EVENTS.Alarms.AlarmsEvent62,1,0);
	GV.stAlarm.Alarm[62].CreateEx(TC_EVENTS.Alarms.AlarmsEvent63,1,0);
	GV.stAlarm.Alarm[63].CreateEx(TC_EVENTS.Alarms.AlarmsEvent64,1,0);
	GV.stAlarm.Alarm[64].CreateEx(TC_EVENTS.Alarms.AlarmsEvent65,1,0);
	GV.stAlarm.Alarm[65].CreateEx(TC_EVENTS.Alarms.AlarmsEvent66,1,0);
	GV.stAlarm.Alarm[66].CreateEx(TC_EVENTS.Alarms.AlarmsEvent67,1,0);
	GV.stAlarm.Alarm[67].CreateEx(TC_EVENTS.Alarms.AlarmsEvent68,1,0);
	GV.stAlarm.Alarm[68].CreateEx(TC_EVENTS.Alarms.AlarmsEvent69,1,0);
	GV.stAlarm.Alarm[69].CreateEx(TC_EVENTS.Alarms.AlarmsEvent70,1,0);
	
END_IF
END_ACTION

ACTION ACT_Raise:
FOR iRaise:=0 TO 69 DO
	IF GV.stAlarm.Raise[iRaise] THEN
		GV.stAlarm.Alarm[iRaise].Raise(0);
	END_IF

END_FOR
END_ACTION

END_PROGRAM

(* stored: Version 1.1.0.1, ProductVersion 3.1.4024.12
   POU P1_04_Alarms: Id {05a3b4e5-763c-4134-adea-e0ffcecea08d}, SpecialFunc None
   Action ACT_Ack: Id {38bcc089-4166-4bc8-8e7d-87cb4ae9c08b}
   Action ACT_Active: Id {03da289e-5970-482e-a297-51b7f8397c80}
   Action ACT_Disabled: Id {c62d7609-3940-46a3-885c-3247e26adbe0}
   Action ACT_Init: Id {181bf5ce-27d5-4fe3-b170-4e8cad8c1884}
   Action ACT_Raise: Id {c0adc887-b8e8-40fe-922b-74f7b64f19fc} *)
